FUNCTION_BLOCK E_PERMIT (* permissive propagation of an event *)
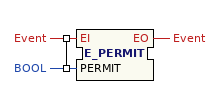
  EVENT_INPUT
    EI WITH PERMIT; (* Event input *)
  END_EVENT
  EVENT_OUTPUT
    EO; (* Event output *)
  END_EVENT
  VAR_INPUT
    PERMIT : BOOL;
  END_VAR
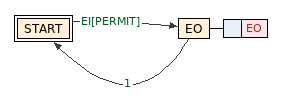
  EC_STATES
    START; (* Initial State *)
    EO : -> EO; (* Event propagration permited *)
  END_STATES
  EC_TRANSITIONS
    START TO EO := EI[PERMIT];
    EO TO START := 1;
  END_TRANSITIONS
END_FUNCTION_BLOCK
